(* PLC project Unnamed, Unknown Unnamed 1 *)
(* stored: creationDateTime 2012-09-12T23:30:19, modificationDateTime 2013-05-16T17:17:49 *)

PROGRAM main
  VAR
    x : INT;
    y : INT;
    b1 : BYTE;
    b0 : BYTE;
  END_VAR
  VAR_EXTERNAL
    WiiNunchuckStickX : INT;
    WiiNunchuckStickY : INT;
    WiiNunchuckButtons : BYTE;
    WiiButtons : BYTE;
  END_VAR

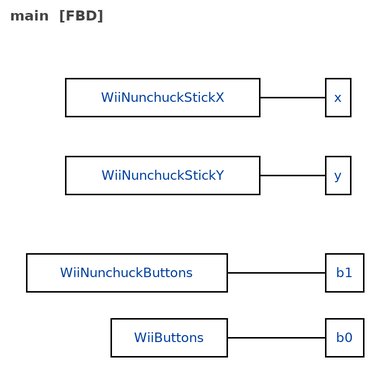
(* FBD diagram, written out as Structured Text *)
x := WiiNunchuckStickX;
y := WiiNunchuckStickY;
b1 := WiiNunchuckButtons;
b0 := WiiButtons;
END_PROGRAM

CONFIGURATION config
  RESOURCE resource1 ON PLC
    TASK tsk1(INTERVAL := T#1ms, PRIORITY := 0);
    PROGRAM inst1 WITH tsk1 : main;
  END_RESOURCE
END_CONFIGURATION
